// Mitsubishi GX Works2 project: TEx01   PLC: Q02/Q02H

PROGRAM MAIN
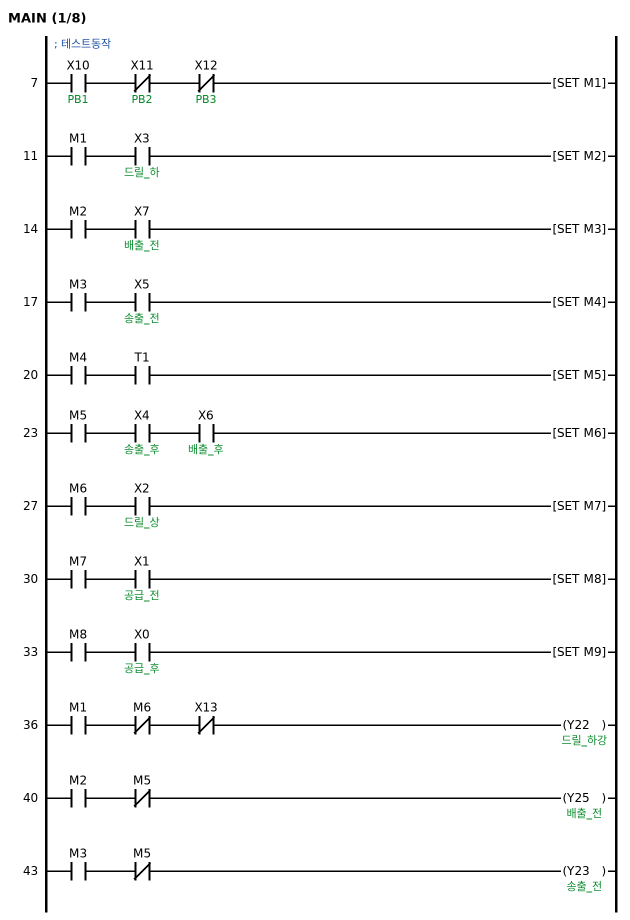
; 테스트동작
7     LD      X10  ; PB1
      ANI     X11  ; PB2
      ANI     X12  ; PB3
      SET     M1
11    LD      M1
      AND     X3  ; 드릴_하
      SET     M2
14    LD      M2
      AND     X7  ; 배출_전
      SET     M3
17    LD      M3
      AND     X5  ; 송출_전
      SET     M4
20    LD      M4
      AND     T1
      SET     M5
23    LD      M5
      AND     X4  ; 송출_후
      AND     X6  ; 배출_후
      SET     M6
27    LD      M6
      AND     X2  ; 드릴_상
      SET     M7
30    LD      M7
      AND     X1  ; 공급_전
      SET     M8
33    LD      M8
      AND     X0  ; 공급_후
      SET     M9
36    LD      M1
      ANI     M6
      ANI     X13
      OUT     Y22  ; 드릴_하강
40    LD      M2
      ANI     M5
      OUT     Y25  ; 배출_전
43    LD      M3
      ANI     M5
      OUT     Y23  ; 송출_전
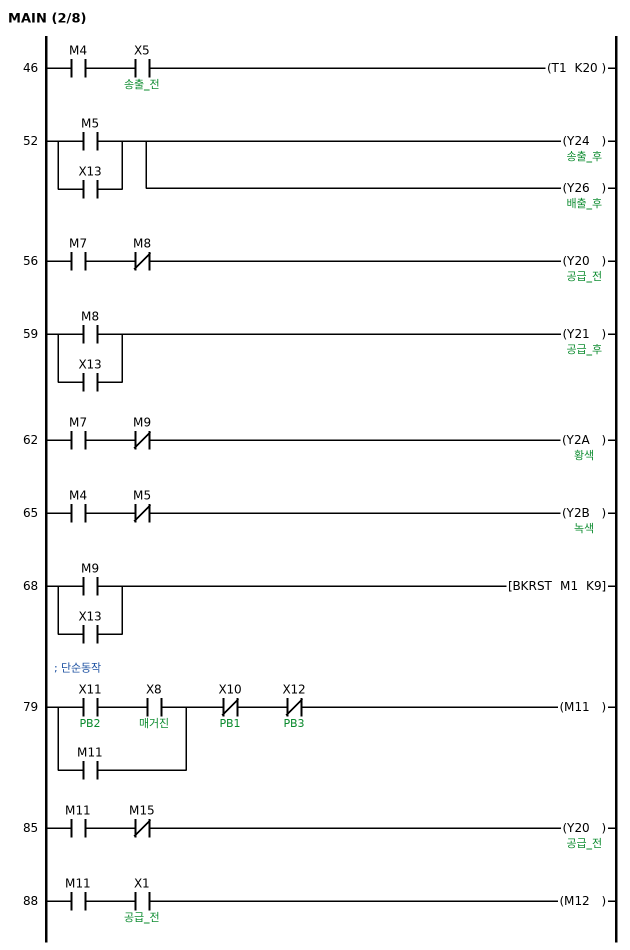
46    LD      M4
      AND     X5  ; 송출_전
      OUT     T1 K20
52    LD      M5
      OR      X13
      OUT     Y24  ; 송출_후
      OUT     Y26  ; 배출_후
56    LD      M7
      ANI     M8
      OUT     Y20  ; 공급_전
59    LD      M8
      OR      X13
      OUT     Y21  ; 공급_후
62    LD      M7
      ANI     M9
      OUT     Y2A  ; 황색
65    LD      M4
      ANI     M5
      OUT     Y2B  ; 녹색
68    LD      M9
      OR      X13
      BKRST   M1 K9
; 단순동작
79    LD      X11  ; PB2
      AND     X8  ; 매거진
      OR      M11
      ANI     X10  ; PB1
      ANI     X12  ; PB3
      OUT     M11
85    LD      M11
      ANI     M15
      OUT     Y20  ; 공급_전
88    LD      M11
      AND     X1  ; 공급_전
      OUT     M12
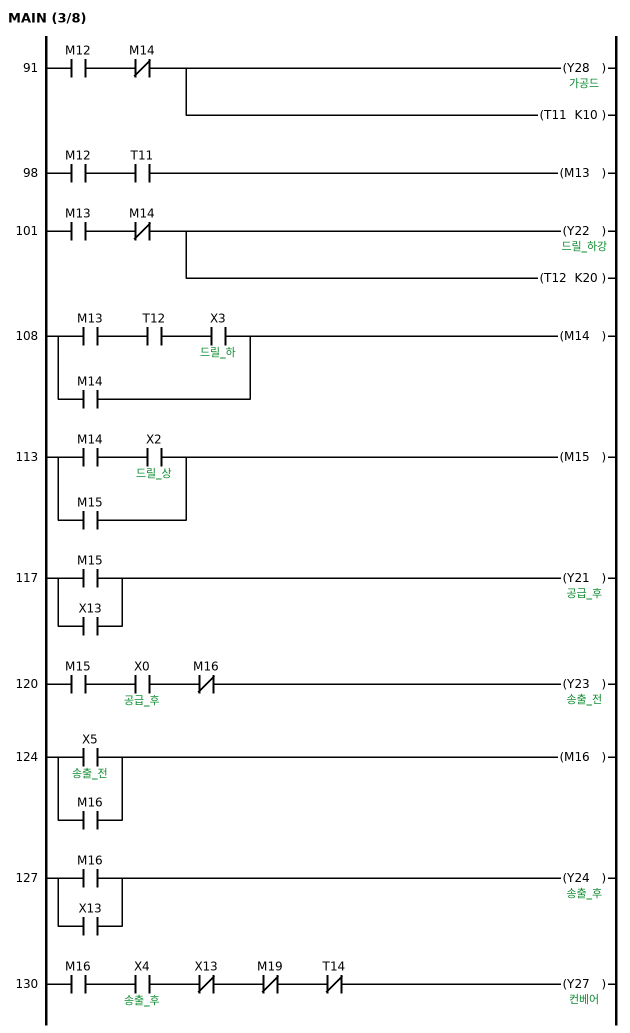
91    LD      M12
      ANI     M14
      OUT     Y28  ; 가공드
      OUT     T11 K10
98    LD      M12
      AND     T11
      OUT     M13
101   LD      M13
      ANI     M14
      OUT     Y22  ; 드릴_하강
      OUT     T12 K20
108   LD      M13
      AND     T12
      AND     X3  ; 드릴_하
      OR      M14
      OUT     M14
113   LD      M14
      AND     X2  ; 드릴_상
      OR      M15
      OUT     M15
117   LD      M15
      OR      X13
      OUT     Y21  ; 공급_후
120   LD      M15
      AND     X0  ; 공급_후
      ANI     M16
      OUT     Y23  ; 송출_전
124   LD      X5  ; 송출_전
      OR      M16
      OUT     M16
127   LD      M16
      OR      X13
      OUT     Y24  ; 송출_후
130   LD      M16
      AND     X4  ; 송출_후
      ANI     X13
      ANI     M19
      ANI     T14
      OUT     Y27  ; 컨베어
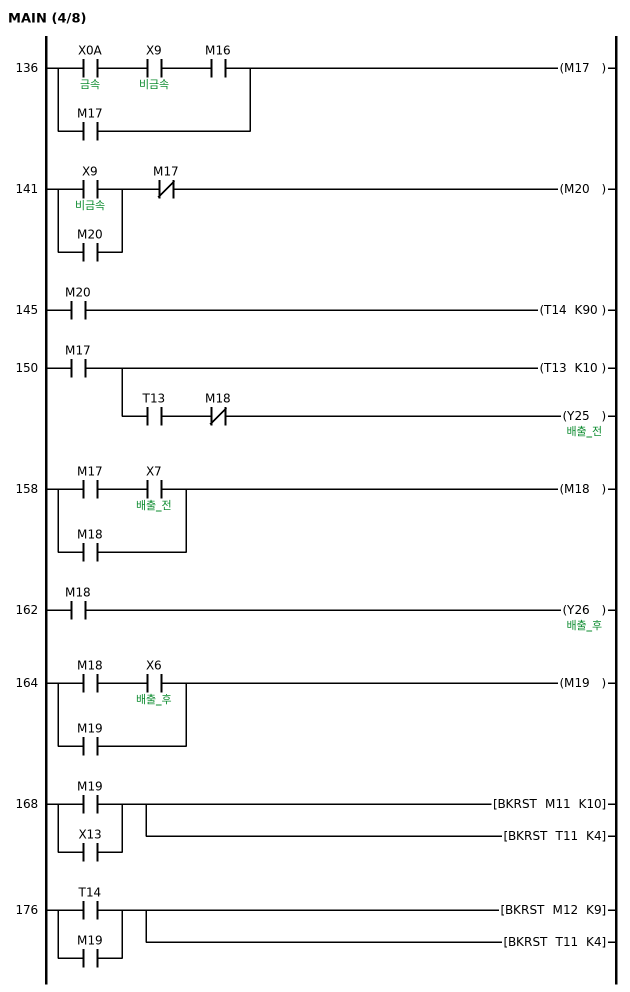
136   LD      X0A  ; 금속
      AND     X9  ; 비금속
      AND     M16
      OR      M17
      OUT     M17
141   LD      X9  ; 비금속
      OR      M20
      ANI     M17
      OUT     M20
145   LD      M20
      OUT     T14 K90
150   LD      M17
      OUT     T13 K10
      AND     T13
      ANI     M18
      OUT     Y25  ; 배출_전
158   LD      M17
      AND     X7  ; 배출_전
      OR      M18
      OUT     M18
162   LD      M18
      OUT     Y26  ; 배출_후
164   LD      M18
      AND     X6  ; 배출_후
      OR      M19
      OUT     M19
168   LD      M19
      OR      X13
      BKRST   M11 K10
      BKRST   T11 K4
176   LD      T14
      OR      M19
      BKRST   M12 K9
      BKRST   T11 K4
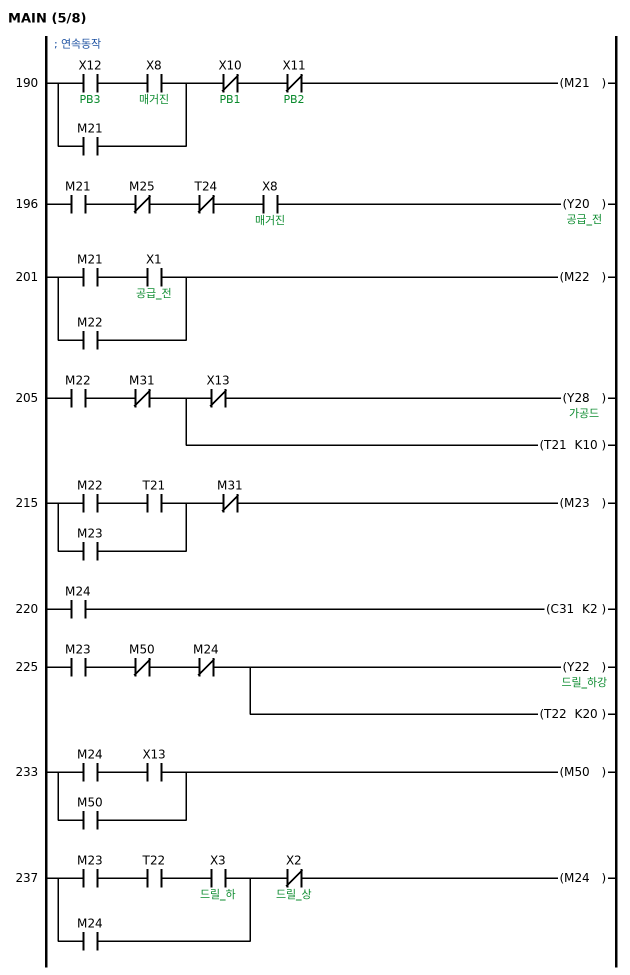
; 연속동작
190   LD      X12  ; PB3
      AND     X8  ; 매거진
      OR      M21
      ANI     X10  ; PB1
      ANI     X11  ; PB2
      OUT     M21
196   LD      M21
      ANI     M25
      ANI     T24
      AND     X8  ; 매거진
      OUT     Y20  ; 공급_전
201   LD      M21
      AND     X1  ; 공급_전
      OR      M22
      OUT     M22
205   LD      M22
      ANI     M31
      MPS
      ANI     X13
      OUT     Y28  ; 가공드
      MPP
      OUT     T21 K10
215   LD      M22
      AND     T21
      OR      M23
      ANI     M31
      OUT     M23
220   LD      M24
      OUT     C31 K2
225   LD      M23
      ANI     M50
      ANI     M24
      OUT     Y22  ; 드릴_하강
      OUT     T22 K20
233   LD      M24
      AND     X13
      OR      M50
      OUT     M50
237   LD      M23
      AND     T22
      AND     X3  ; 드릴_하
      OR      M24
      ANI     X2  ; 드릴_상
      OUT     M24
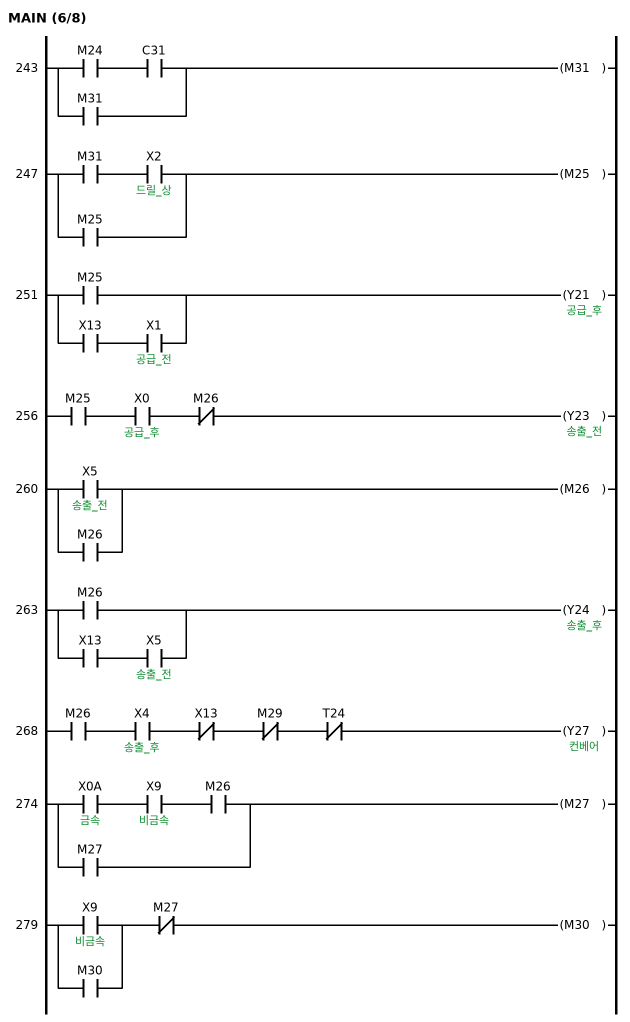
243   LD      M24
      AND     C31
      OR      M31
      OUT     M31
247   LD      M31
      AND     X2  ; 드릴_상
      OR      M25
      OUT     M25
251   LD      M25
      LD      X13
      AND     X1  ; 공급_전
      ORB
      OUT     Y21  ; 공급_후
256   LD      M25
      AND     X0  ; 공급_후
      ANI     M26
      OUT     Y23  ; 송출_전
260   LD      X5  ; 송출_전
      OR      M26
      OUT     M26
263   LD      M26
      LD      X13
      AND     X5  ; 송출_전
      ORB
      OUT     Y24  ; 송출_후
268   LD      M26
      AND     X4  ; 송출_후
      ANI     X13
      ANI     M29
      ANI     T24
      OUT     Y27  ; 컨베어
274   LD      X0A  ; 금속
      AND     X9  ; 비금속
      AND     M26
      OR      M27
      OUT     M27
279   LD      X9  ; 비금속
      OR      M30
      ANI     M27
      OUT     M30
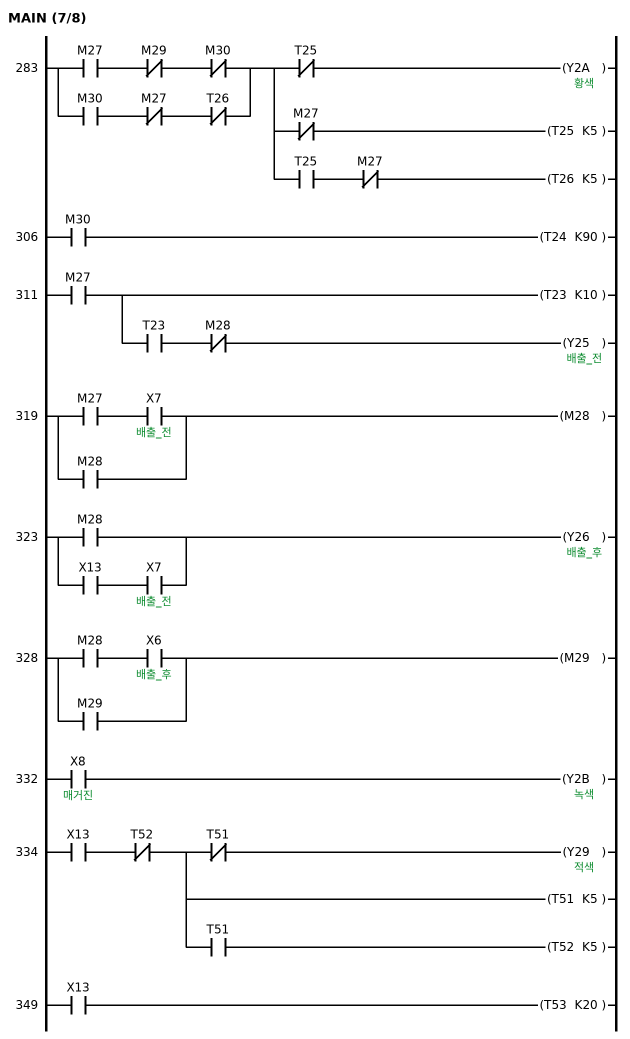
283   LD      M27
      ANI     M29
      ANI     M30
      LD      M30
      ANI     M27
      ANI     T26
      ORB
      MPS
      ANI     T25
      OUT     Y2A  ; 황색
      MRD
      ANI     M27
      OUT     T25 K5
      MPP
      AND     T25
      ANI     M27
      OUT     T26 K5
306   LD      M30
      OUT     T24 K90
311   LD      M27
      OUT     T23 K10
      AND     T23
      ANI     M28
      OUT     Y25  ; 배출_전
319   LD      M27
      AND     X7  ; 배출_전
      OR      M28
      OUT     M28
323   LD      M28
      LD      X13
      AND     X7  ; 배출_전
      ORB
      OUT     Y26  ; 배출_후
328   LD      M28
      AND     X6  ; 배출_후
      OR      M29
      OUT     M29
332   LD      X8  ; 매거진
      OUT     Y2B  ; 녹색
334   LD      X13
      ANI     T52
      MPS
      ANI     T51
      OUT     Y29  ; 적색
      MPP
      OUT     T51 K5
      AND     T51
      OUT     T52 K5
349   LD      X13
      OUT     T53 K20
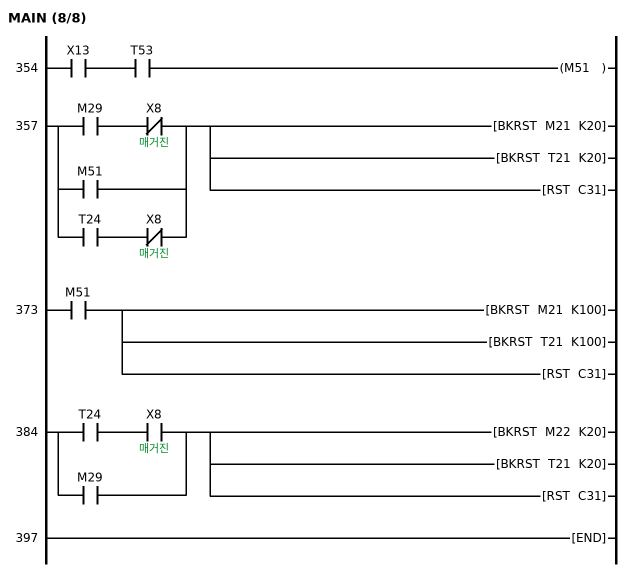
354   LD      X13
      AND     T53
      OUT     M51
357   LD      M29
      ANI     X8  ; 매거진
      OR      M51
      LD      T24
      ANI     X8  ; 매거진
      ORB
      BKRST   M21 K20
      BKRST   T21 K20
      RST     C31
373   LD      M51
      BKRST   M21 K100
      BKRST   T21 K100
      RST     C31
384   LD      T24
      AND     X8  ; 매거진
      OR      M29
      BKRST   M22 K20
      BKRST   T21 K20
      RST     C31
397   END
END_PROGRAM
